// TIA Portal V17 export
// export: Created 2022-07-20T06:59:42.4462973Z, ExportSetting WithDefaults, DisplayName Totally Integrated Automation Portal, DisplayVersion V17, DisplayName TIA Portal Openness, DisplayVersion V17, DisplayName TIA Portal Version Control Interface, DisplayVersion V17, DisplayName SINAMICS Startdrive Advanced, DisplayVersion V17, DisplayName SINAMICS Startdrive G130, G150, S120, S150, SINAMICS MV, S210, DisplayVersion V17, DisplayName SINAMICS Startdrive G110M, G120, G120C, G120D, G120P, G115D, DisplayVersion V17, DisplayName STEP 7 Professional, DisplayVersion V17, DisplayName STEP 7 Safety, DisplayVersion V17, DisplayName WinCC Advanced, DisplayVersion V17
FUNCTION_BLOCK "FB10072_AirExtractorAnalogManager"   // FB10072, LAD
TITLE = FB10072_AirExtractorAnalogManager
{ S7_Optimized_Access := 'TRUE' }
AUTHOR : Jonathan
FAMILY : 1007x_DRYER_UV
VERSION : 1.0
// Release note : 
// 1.0 - Feature developped
// stored: AutoNumber false, IsIECCheckEnabled false, IsRetainMemResEnabled false, MemoryReserve 100, SetENOAutomatically false, UDAEnableTagReadback false
   VAR_INPUT
      UVReady : Bool;
      UVFeedbackPower : Real;
      UVEnabled : Bool;
      AirExtractionActivation : Bool;
      ForceAirAfterShutdownUV : Bool;
      ShutterOpen : Bool;
      ShutterClose : Bool;
      ScalingShutterOpen : "stAirExtractorScalingParameters";
      ScalingShutterClosed : "stAirExtractorScalingParameters";
   END_VAR
   VAR_OUTPUT
      AirExtractionEnable : Bool;
      AirExractionAnalogPowerValue : Int;
      ForcingAirInProgress : Bool;
   END_VAR
   VAR
      CoolingAfterClosing : Bool;
      RTrig_ShutterClose { S7_SetPoint := 'True'} : R_TRIG;
      RTrig_ForceAir { S7_SetPoint := 'True'} : R_TRIG;
      TOF_ForceAirTimer { S7_SetPoint := 'True'} : TOF_TIME;
      MemUVEnabledOnce : Bool;
   END_VAR
   VAR_TEMP
      temp_real : Real;
   END_VAR
BEGIN

REGION Network 1 (SCL): Scale Dryer Uv Power Calculation
   // Rising edge shutter closed
   #RTrig_ShutterClose(CLK := #ShutterClose);
   // Force cooling until UV Ready
   IF #RTrig_ShutterClose.Q THEN
       #CoolingAfterClosing := TRUE;
   END_IF;

   // Reset cooling if UV Ready
   IF (#UVFeedbackPower/276.48) <= #ScalingShutterClosed.PowerXMin THEN
       #CoolingAfterClosing := FALSE;
   END_IF;

   // Memorisation if UV was enabled one time at least
   IF #UVEnabled THEN
       #MemUVEnabledOnce := TRUE;
   END_IF;

   IF #TOF_ForceAirTimer.Q THEN
       #MemUVEnabledOnce := FALSE;
       #ForcingAirInProgress := TRUE;
   ELSE
       #ForcingAirInProgress := FALSE;
   END_IF;

   // Rising edge on force Air
   #RTrig_ForceAir(CLK := #ForceAirAfterShutdownUV);
   #TOF_ForceAirTimer(IN := #RTrig_ForceAir.Q AND #MemUVEnabledOnce,
                      PT := T#5m);

   // Air Extraction enable
   IF (#AirExtractionActivation AND #UVReady) OR #TOF_ForceAirTimer.Q THEN
       #AirExtractionEnable := TRUE;
   ELSE
       #AirExtractionEnable := FALSE;
   END_IF;


   // Scaling 
   IF #CoolingAfterClosing OR #TOF_ForceAirTimer.Q THEN
       // Force cooling after closing until UV Ready or After shutdown UV
       #AirExractionAnalogPowerValue := 27648;
   ELSIF  #ShutterClose AND #AirExtractionEnable THEN
       "FC10070_ScalingAirExtraction"(SetPoint := (#UVFeedbackPower/276.48),
                                     X_UVPower_Min := #ScalingShutterClosed.PowerXMin,
                                     X_UVPower_Max := #ScalingShutterClosed.PowerXMax,
                                     Y_AirPower_Min := #ScalingShutterClosed.PowerAirYMin,
                                     Y_AirPower_Max := #ScalingShutterClosed.PowerAirYMax,
                                     PWM_Minimum:= 0.0,
                                     PWM_Maximum:= 100.0,
                                     AnalogValue => #AirExractionAnalogPowerValue,
                                     PwmFrequenceValue=>#temp_real);
   ELSIF #ShutterOpen AND #AirExtractionEnable THEN
       "FC10070_ScalingAirExtraction"(SetPoint := (#UVFeedbackPower/276.48),
                                     X_UVPower_Min := #ScalingShutterOpen.PowerXMin,
                                     X_UVPower_Max := #ScalingShutterOpen.PowerXMax,
                                     Y_AirPower_Min := #ScalingShutterOpen.PowerAirYMin,
                                     Y_AirPower_Max := #ScalingShutterOpen.PowerAirYMax,
                                     PWM_Minimum:= 0.0 ,
                                     PWM_Maximum:= 100.0,
                                     AnalogValue => #AirExractionAnalogPowerValue,
                                     PwmFrequenceValue=>#temp_real);
   ELSE
       #AirExractionAnalogPowerValue := 0;
   END_IF;
END_REGION
END_FUNCTION_BLOCK
